(* PLC project v0.6.04_CycleSemiAuto.project, CODESYS CODESYS V3.5 SP19 Patch 1 *)
(* stored: creationDateTime 2026-08-17T05:53:47.249603, modificationDateTime 2026-08-17T05:53:47.249603 *)

(* ═══════════════════════════════════════════════════════════════ 🔧 ST_DredgingAssistCfg — Réglages persistants assistants prélèvement 📄 Doc : DOC/AF/AF_Partie-04_Mode_SemiAuto_Sequenceur_v2.1.md §3ter ═══════════════════════════════════════════════════════════════ *)
TYPE ST_DredgingAssistCfg : STRUCT
  DiveStartMin_M : REAL := 1;  (* Position mini M1/M2 avant plongée *)
  ImmersionUpper_M : REAL := 0.5;  (* Borne haute fenêtre front immersion *)
  ImmersionLower_M : REAL := -0.5;  (* Borne basse fenêtre front immersion *)
  ExtractionControlDistance_M : REAL := 2;  (* Remontée palier 1 avant accélération *)
  TglEnableDiveSearch : BOOL := TRUE;  (* Mode assistance plongée mémorisé *)
  TglEnableExtractionSequence : BOOL := TRUE;  (* Mode assistance extraction mémorisé *)
  TglEnableDumpAtTremie : BOOL := TRUE;  (* Mode assistance vidage trémie mémorisé *)
  Initialized : BOOL := FALSE;  (* Pont persistance/IHM initialisé *)
END_STRUCT;
END_TYPE
